SUBAPPLICATION Uebung_006a (* SR und T-Flip-Flop mit 3x IE *)
  (* Standard: 61499-2; Description: Copyright (c) 2023 Meisterschulen am Ostbahnhof This program and the accompanying materials are made available under the terms of the Eclipse Public License 2.0 which is available at https://www.eclipse.org/legal/epl-2.0/ SPDX-License-Identifier: EPL-2.0 *)
  (* Version 1.0, 2023-10-23, Franz Höpfinger, Meisterschulen am Ostbahnhof *)
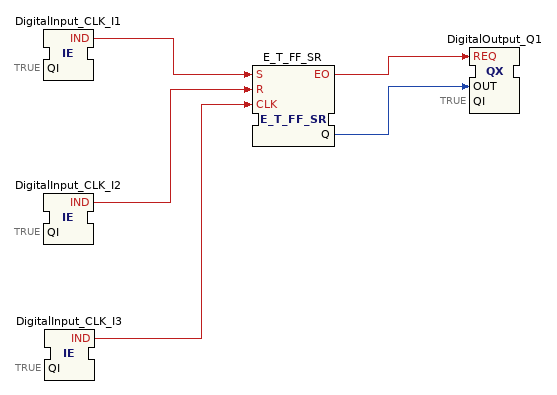
  FBS
    DigitalOutput_Q1 : QX(QI := TRUE);
    DigitalInput_CLK_I1 : IE(QI := TRUE);
    DigitalInput_CLK_I2 : IE(QI := TRUE);
    E_T_FF_SR : E_T_FF_SR;
    DigitalInput_CLK_I3 : IE(QI := TRUE);
  END_FBS
  EVENT_CONNECTIONS
    DigitalInput_CLK_I1.IND TO E_T_FF_SR.S;
    DigitalInput_CLK_I2.IND TO E_T_FF_SR.R;
    E_T_FF_SR.EO TO DigitalOutput_Q1.REQ;
    DigitalInput_CLK_I3.IND TO E_T_FF_SR.CLK;
  END_CONNECTIONS
  DATA_CONNECTIONS
    E_T_FF_SR.Q TO DigitalOutput_Q1.OUT;
  END_CONNECTIONS
END_SUBAPPLICATION
